(* IEC 61131-3 sources: sigmatek-logger-api/IXON_API/Class/File_IO, 1 file *)

(* ---- File_IO.st ---- *)
(*!
<Class
	Name               = "File_IO"
	Revision           = "0.1"
	RealtimeTask       = "false"
	CyclicTask         = "false"
	BackgroundTask     = "false"
	Sigmatek           = "true"
	OSInterface        = "true"
	HighPriority       = "false"
	Automatic          = "false"
	UpdateMode         = "Prescan"
	IconPath           = ".\Class\File_IO\Files 1.ico"
	SharedCommandTable = "true"
	Objectsize         = "(284,120)"
	Comment            = "various file-operations like open, close, seek, read and write">
	<Channels>
		<Server Name="Server0" Visualized="true" Initialize="false" WriteProtected="true" Retentive="false"/>
	</Channels>
	<Dependencies>
		<Files>
			<File Path=".\Source\code\OsiBase.h" Include="false"/>
			<File Path=".\File_IOTypes.h" Include="false"/>
			<File Path=".\Source\code\OsiBase.st"/>
		</Files>
	</Dependencies>
</Class>
*)
File_IO : CLASS
  //Servers:
	Server0 	: SvrChCmd_DINT;
  //Clients:
  //Variables:
  //Functions:

	FUNCTION File_IO
		VAR_OUTPUT
			ret_code 	: ConfStates;
		END_VAR;

	FUNCTION __CDECL VIRTUAL GLOBAL FileRead
		VAR_INPUT
			handle 	: DINT;
			data 	: ^void;
			size 	: UDINT;
		END_VAR
		VAR_OUTPUT
			retcode (EAX) 	: UDINT;
		END_VAR;

	FUNCTION __CDECL VIRTUAL GLOBAL FileWrite
		VAR_INPUT
			handle 	: DINT;
			data 	: ^void;
			size 	: UDINT;
		END_VAR
		VAR_OUTPUT
			retcode (EAX) 	: UDINT;
		END_VAR;

	FUNCTION __CDECL VIRTUAL GLOBAL FileOpen
		VAR_INPUT
			path 	: ^CHAR;
			create 	: DINT;
			Attribs 	: UDINT;
		END_VAR
		VAR_OUTPUT
			retcode (EAX) 	: DINT;
		END_VAR;

	FUNCTION __CDECL VIRTUAL GLOBAL FileClose
		VAR_INPUT
			handle 	: DINT;
		END_VAR;

	FUNCTION __CDECL VIRTUAL GLOBAL FileDelete
		VAR_INPUT
			file 	: ^CHAR;
		END_VAR
		VAR_OUTPUT
			retcode (EAX) 	: DINT;
		END_VAR;

	FUNCTION __CDECL VIRTUAL GLOBAL FilelSeek
		VAR_INPUT
			handle 	: DINT;
			offset 	: UDINT;
			fromwhere 	: UDINT;
		END_VAR
		VAR_OUTPUT
			retcode (EAX) 	: UDINT;
		END_VAR;

	FUNCTION __CDECL VIRTUAL GLOBAL FileTell
		VAR_INPUT
			handle 	: DINT;
		END_VAR
		VAR_OUTPUT
			retcode (EAX) 	: DINT;
		END_VAR;

	FUNCTION __CDECL VIRTUAL GLOBAL FileLength
		VAR_INPUT
			handle 	: DINT;
		END_VAR
		VAR_OUTPUT
			retcode (EAX) 	: DINT;
		END_VAR;

	FUNCTION __CDECL VIRTUAL GLOBAL CreateDir
		VAR_INPUT
			name 	: ^CHAR;
		END_VAR
		VAR_OUTPUT
			retcode (EAX) 	: DINT;
		END_VAR;

	FUNCTION __CDECL VIRTUAL GLOBAL RemoveDir
		VAR_INPUT
			name 	: ^CHAR;
		END_VAR
		VAR_OUTPUT
			retcode (EAX) 	: DINT;
		END_VAR;

	FUNCTION __CDECL VIRTUAL GLOBAL FindFirst
		VAR_INPUT
			path 	: ^CHAR;
			fname 	: ^CHAR;
			finfo 	: ^_DDE_INFO;
			att_incl 	: USINT;
			att_excl 	: USINT;
		END_VAR
		VAR_OUTPUT
			retcode (EAX) 	: DINT;
		END_VAR;

	FUNCTION __CDECL VIRTUAL GLOBAL FindNext
		VAR_INPUT
			handle 	: DINT;
			fInfo 	: ^_DDE_INFO;
		END_VAR
		VAR_OUTPUT
			retcode (EAX) 	: DINT;
		END_VAR;

	FUNCTION __CDECL VIRTUAL GLOBAL FindClose
		VAR_INPUT
			handle 	: DINT;
		END_VAR
		VAR_OUTPUT
			retcode (EAX) 	: DINT;
		END_VAR;

	FUNCTION __CDECL VIRTUAL GLOBAL CloseAllOpenFiles;

	FUNCTION __CDECL VIRTUAL GLOBAL Rename
		VAR_INPUT
			oldname 	: ^CHAR;
			newname 	: ^CHAR;
		END_VAR
		VAR_OUTPUT
			retcode (EAX) 	: DINT;
		END_VAR;
  //Tables:
	FUNCTION @STD
		VAR_OUTPUT
			ret_code	: CONFSTATES;
		END_VAR;
	FUNCTION GLOBAL TAB @CT_;
END_CLASS;

//*********************Inserted from .\code\File_IO.st*********************

#include "..\..\Source\code\OsiBase.h"

FUNCTION  File_IO::File_IO
VAR_OUTPUT
	ret_code		: CONFSTATES;
END_VAR

	ret_code	:= InitOsiM(_lsl_pOS^.piFILE, USER_CNT_File_IO);

END_FUNCTION // File_IO::File_IO
